FUNCTION_BLOCK FB_NormalWash IMPLEMENTS I_WashStrategy
VAR
	 bStarted : BOOL := FALSE; 
	 stSettings : ST_WashSettings;
END_VAR

METHOD FB_init : BOOL
VAR_INPUT
	bInitRetains : BOOL; // if TRUE, the retain variables are initialized (warm start / cold start)
	bInCopyCode : BOOL;  // if TRUE, the instance afterwards gets moved into the copy code (online change)
END_VAR
stSettings.rTemperature  := GVL_WashConstants.NORMAL_TEMP; 
stSettings.nSpinSpeed    := GVL_WashConstants.NORMAL_SPIN; 
stSettings.tWashDuration := GVL_WashConstants.NORMAL_WASH_TIME; 
stSettings.sDescription  := GVL_WashConstants.NORMAL_DESC; 

FB_init := TRUE;
END_METHOD

METHOD GetDuration : TIME
GetDuration := stSettings.tWashDuration;
END_METHOD

METHOD GetProgramName : STRING
GetProgramName := 'NORMAL';
END_METHOD

METHOD GetSettings : ST_WashSettings
GetSettings := stSettings;
END_METHOD

METHOD Start : BOOL
bStarted := TRUE; 
Start     := TRUE;
END_METHOD

END_FUNCTION_BLOCK

(* stored: Version 1.1.0.1, ProductVersion 3.1.4024.16
   POU FB_NormalWash: Id {1a40042c-adbf-4b51-8b38-404cab057683}, SpecialFunc None
   Method FB_init: Id {f1536ea9-43f7-4a5e-a2e1-5f4c5af6adcb}
   Method GetDuration: Id {7a82bdcf-7c45-449f-b64f-7b4116fa5130}
   Method GetProgramName: Id {2bc7e14b-0b7b-471c-a067-5f9298e74cf0}
   Method GetSettings: Id {940ca7a1-1be0-4abc-b0f9-cd30c21e2f50}
   Method Start: Id {d6ca3d32-fd76-4dee-b80c-59ece26bcca3} *)
